(* CODESYS project Minimalbeispiel_Datenaustausch_ROS2_OPCUA.project

Project tree, tasks and I/O mapping:
  Device : CODESYS Virtual Control for Linux SL, CODESYS, order no. 2302000005, version 4.22.0.0
    application Application
      task MainTask (cyclic, interval t#20ms, priority 1) calls PLC_PRG
      task VISU_TASK (cyclic, interval 100 ms, priority 31) calls VisuElems.Visu_Prg
      program PLC_PRG [ST]
      Kommunikationsverwalter
        OPC UA Server
          Symbolgruppe
      global variables GVL_OPCUA
      data type turtlesim_msg_pose
      visualisation Visualization
      data type geometry_msgs_msg_Twist
      data type turtlesim_srv_Spawn
      Symbols
  libraries: SM3_Robotics, * (CODESYS); VisuSymbols, 4.5.0.0 (System)
  text list GlobalTextList
*)

// Device/Application/turtlesim_msg_pose
TYPE turtlesim_msg_pose :
STRUCT
	x_pose : REAL;			
	y_pose : REAL;			
	theta_pose : REAL;		//in RAD
	linear_velocity_pose : REAL;	
	angular_velocity_pose : REAL;	
END_STRUCT
END_TYPE

// Device/Application/geometry_msgs_msg_Twist
TYPE geometry_msgs_msg_Twist :
STRUCT
	linear_x : LREAL;
	linear_y : LREAL;
	linear_z : LREAL;
	
	angular_x : LREAL;
	angular_y : LREAL;
	angular_z : LREAL;
END_STRUCT
END_TYPE

// Device/Application/turtlesim_srv_Spawn
TYPE turtlesim_srv_Spawn :
STRUCT
	//SPS -> ROS2
	xExecute : BOOL;
	req_x : REAL;
	req_y : REAL;
	req_theta : REAL;
	req_name : STRING;
	//ROS2 -> SPS
	xDone : BOOL;
	xError : BOOL;
	resp_name : STRING;
END_STRUCT
END_TYPE

// Device/Application/GVL_OPCUA
{attribute 'qualified_only'}
VAR_GLOBAL
	PI : REAL := 3.14159;

	//Datenaustausch CODESYS -> ROS2
	turtle1_cmd_vel : geometry_msgs_msg_Twist;	//topic: /turtle1/cmd_vel mit interface geometry_msgs/msg/Twist
	//Datenaustausch ROS2 -> CODESYS
	turtle1_pose : turtlesim_msg_pose;			//topic: /turtle1/pose mit interface turlesim/msg/Pose
	
	//Service 
	spawn : turtlesim_srv_Spawn;				//service: /spawn mit interface turtlesim/srv/Spawn
	
END_VAR

// Device/Application/PLC_PRG
PROGRAM PLC_PRG
VAR
	// /turtle1/pos
	theta_deg : REAL;
	y_negative : REAL;
	x_normal: REAL;
	
	vor : BOOL := FALSE;
	rueck : BOOL := FALSE;
	links : BOOL := FALSE;
	rechts : BOOL := FALSE;
	
END_VAR

// Für Visualisierung skalieren
theta_deg := - GVL_OPCUA.turtle1_pose.theta_pose * (180.0/3.14159);
y_negative := - GVL_OPCUA.turtle1_pose.y_pose *(300/11.088);
x_normal := GVL_OPCUA.turtle1_pose.x_pose * (300/11.088);

// Buttons für Visualisierung
IF vor = TRUE THEN
	GVL_OPCUA.turtle1_cmd_vel.linear_x := 0.6;

ELSIF rueck = TRUE THEN
	GVL_OPCUA.turtle1_cmd_vel.linear_x := -0.6;
	
ELSIF rechts = TRUE THEN
	GVL_OPCUA.turtle1_cmd_vel.angular_z := - 0.6;

ELSIF links = TRUE THEN
	GVL_OPCUA.turtle1_cmd_vel.angular_z := 0.6;	
ELSE
	GVL_OPCUA.turtle1_cmd_vel.angular_z := 0.0;
	GVL_OPCUA.turtle1_cmd_vel.linear_x := 0.0;
END_IF

END_PROGRAM

// Device/Application/Visualization
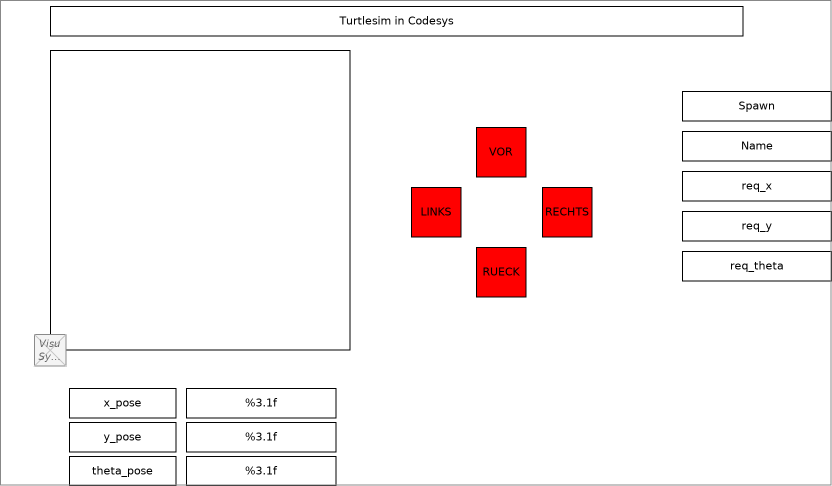
VISUALIZATION Visualization  // 832x486
    Rectangle (50,50 300x300)
    Rectangle (186,388 150x30), "%3.1f", text variable: GVL_OPCUA.turtle1_pose.x_pose
    Rectangle (69,388 107x30), "x_pose"
    Rectangle (69,422 107x30), "y_pose"
    Rectangle (69,456 107x30), "theta_pose", text variable: GVL_OPCUA.turtle1_pose.theta_pose
    Rectangle (186,422 150x30), "%3.1f", text variable: GVL_OPCUA.turtle1_pose.y_pose
    Rectangle (186,456 150x30), "%3.1f", text variable: GVL_OPCUA.turtle1_pose.theta_pose
    Image (34,334 32x32), image: VisuSymbols.Symbols.ArrowBoldRight
        p3560616238: PLC_PRG.x_normal
        p2738717112: PLC_PRG.y_negative
        p2858320360: PLC_PRG.theta_deg
    Rectangle (476,127 50x50), "VOR"
        tap PLC_PRG.vor
    Rectangle (476,247 50x50), "RUECK"
        tap PLC_PRG.rueck
    Rectangle (542,187 50x50), "RECHTS"
        tap PLC_PRG.rechts
    Rectangle (411,187 50x50), "LINKS"
        tap PLC_PRG.links
    Rectangle (50,6 693x30), "Turtlesim in Codesys"
    Rectangle (682,91 150x30), "Spawn"
    Rectangle (682,131 150x30), "Name"
    Rectangle (682,171 150x30), "req_x"
    Rectangle (682,211 150x30), "req_y"
    Rectangle (682,251 150x30), "req_theta"
END_VISUALIZATION
